{attribute 'GeneratedUsingTerminal: EL2595-0000-0018'}
{attribute addProperty BoxType "EL2595-0000-0018"}
{attribute addProperty Id "OutputBOOL1Input_trigger_enableBOOL1ResetBOOL1"}
{attribute addProperty CRC "1984492594"}
{attribute addProperty Size "3"}
TYPE Control_7648F432 :
STRUCT
	{attribute addProperty Name "Output"}
	Output : BOOL;
	{attribute addProperty Name "Input_trigger_enable"}
	Input_trigger_enable : BOOL;
	{attribute addProperty Name "Reset"}
	Reset : BOOL;
END_STRUCT
END_TYPE

(* stored: Version 1.2.0.0, ProductVersion 3.1.4024.9
   DUT Control_7648F432: Id {fdf1941b-f97e-45ad-b413-1a8f40b3beaa} *)
